PROGRAM MAIN
VAR
END_VAR

END_PROGRAM

(* stored: Version 1.1.0.1
   POU MAIN: Id {15583e3e-071e-4372-a61e-f5efc5be48d6} *)
